(* PLC project Generated.project, CODESYS CODESYS V3.5 SP19 Patch 1 *)
(* stored: creationDateTime 2026-08-26T16:40:01.127490, modificationDateTime 2026-08-26T16:40:01.127490 *)

(* ======================================================================= ⚙️ ST_Safety_Emergency_InternalCmd — Structure de commande interne ─────────────────────────────────────────────────────────────── 🎯 Rôle : Transporte les ordres logiques entre le bloc de décision et de sortie AU 🔒 Polarité : MaintainA/B_Cmd en maintien (TRUE = voie saine) 📄 Doc métier : DOC/AF/AF_Partie-01_Analyse_Fonctionnelle_v2.1.md ======================================================================= *)
TYPE ST_Safety_Emergency_InternalCmd : STRUCT
  MaintainA_Cmd : BOOL;  (* Ordre maintien canal A (TRUE = voie maintenue, FALSE = coupure demandee) *)
  MaintainB_Cmd : BOOL;  (* Ordre maintien canal B (TRUE = voie maintenue, FALSE = coupure demandee) *)
  ArmPulse_Cmd : BOOL;  (* Ordre impulsion de rearmement (TRUE = bobine rearmement activee) *)
END_STRUCT;
END_TYPE
